	(*Zjeżdzam na osią pionową Z na pozycję chwytania i załączam ssawki*)		
	E_CapPreScrewer.ePicking:
		//Podjedź robotem w górę	
		mcCartesianZMoveAbsolute.Execute			:= TRUE;		
		mcCartesianZMoveAbsolute.Position			:= stParameters.lrPickZPosition;
		mcCartesianZMoveAbsolute.Acceleration		:= stParameters.lrPickerAcceleration;
		mcCartesianZMoveAbsolute.Deceleration		:= stParameters.lrPickerAcceleration;
		mcCartesianZMoveAbsolute.Velocity			:= stParameters.lrPickerSpeed;
		//Czekam na wykonanie ruchu
		IF mcCartesianZMoveAbsolute.Done THEN
			//Reset komendy ruchu osi
			mcCartesianZMoveAbsolute.Execute		:= FALSE;
			
			//Zeruje rejestry oraz załączanie ssawek
			 FOR i:=1 TO 4 DO
				 bCapSucker[i]						:= stParameters.bPickerActiv[i]; 
				 aCapPresence[i] 					:= FALSE;
			 END_FOR
	
			//Następny krok
			eRunningState							:= E_CapPreScrewer.eVacumCheckPart1;
		END_IF
	
	(*Sprawdzam czy zassane i jazda w górę*)	
	E_CapPreScrewer.eVacumCheckPart1:
		
		tonVacuumWatchdog.IN						:= TRUE;
		
		IF tonSuckedOk[1].Q = stParameters.bPickerActiv[1] AND tonSuckedOk[2].Q = stParameters.bPickerActiv[2]
			AND tonSuckedOk[3].Q = stParameters.bPickerActiv[3] AND tonSuckedOk[4].Q = stParameters.bPickerActiv[4] THEN
			tonVacuumWatchdog.IN					:= FALSE;
		
				FOR i:=1 TO 4 DO
					IF stParameters.bPickerActiv[i] AND stParameters.bStrawCatcherON AND NOT stMoverStatus.stSlotStatus[i].bTubePresent THEN
						bReject								:= TRUE;
						bTubeReject							:= TRUE;
						lrAxisZ_RejectOffset				:= 0.0;
					END_IF

					IF bMover1InPlacePos THEN
						diMover1VacuumRetry[i]		:= 0;
					ELSE
						diMover2VacuumRetry[i]		:= 0;
					END_IF	
				END_FOR 
				
			eRunningState 							:= E_CapPreScrewer.eVacumCheckPart2;
	
		ELSIF tonVacuumWatchdog.Q THEN
		
			FOR i:=1 TO 4 DO
				bCapSucker[i]							:= tonSuckedOk[i].Q;
				
				//robimy odrzut jeżeli zostanie wykryto brak słomki
				IF stParameters.bPickerActiv[i] AND stParameters.bStrawCatcherON AND NOT stMoverStatus.stSlotStatus[i].bTubePresent THEN
					bReject								:= TRUE;
					bTubeReject							:= TRUE;
					lrAxisZ_RejectOffset				:= 0.0;
				END_IF
				
						//Detekcja niepobranej nasadki --> odrzut aktywowany opcjonalnie z receptury
					IF stParameters.bPickerActiv[i] AND NOT tonSuckedOk[i].Q AND NOT stParameters.bVacuumDeactivate THEN
						bReject							:= SEL(stParameters.bRejectON, bReject, TRUE);
						lrAxisZ_RejectOffset			:= SEL(stParameters.bRejectON, lrAxisZ_RejectOffset, 13.0);	//offset dodatkowego zjazdu kartezjanem 
						
						IF bMover1InPlacePos THEN
							diMover1VacuumRetry[i]		:= diMover1VacuumRetry[i] + 1;
						ELSE	
							diMover2VacuumRetry[i]		:= diMover2VacuumRetry[i] + 1;
						END_IF
					ELSIF tonSuckedOk[i].Q OR stParameters.bVacuumDeactivate THEN
						IF 	bMover1InPlacePos THEN
							diMover1VacuumRetry[i]		:= 0;
						ELSE
							diMover2VacuumRetry[i]		:= 0;
						END_IF	
					END_IF	
	    	
			END_FOR
				tonVacuumWatchdog.IN					:= FALSE;
				eRunningState 							:= E_CapPreScrewer.eVacumCheckPart2;
	
		END_IF
		
		
	E_CapPreScrewer.eVacumCheckPart2:	
			
		//Jezeli nie jest przyssana zadna nasadka to pdjezdzamy na poz. ready oraz wystawiamy flage bMissingCaps
		IF bReject THEN
			Reject();
				IF bRejectDone THEN				
					eRunningState						:= E_CapPreScrewer.eReady;	
				END_IF		
		ELSIF NOT tonSuckedOk[1].Q AND NOT tonSuckedOk[2].Q AND NOT tonSuckedOk[3].Q AND NOT tonSuckedOk[4].Q THEN
			bCapSucker[1]							:= FALSE;
			bCapSucker[2]							:= False;
			bCapSucker[3]							:= False;
		    bCapSucker[4]							:= False;	
			mcCartesianZMoveAbsolute.Execute		:= TRUE;		
			mcCartesianZMoveAbsolute.Position		:= stParameters.lrTopZPosition;
			mcCartesianZMoveAbsolute.Acceleration	:= stParameters.lrPickerAcceleration;
			mcCartesianZMoveAbsolute.Deceleration	:= stParameters.lrPickerAcceleration;
			mcCartesianZMoveAbsolute.Velocity		:= stParameters.lrPickerSpeed;
			
			IF mcCartesianZMoveAbsolute.Done THEN
				bMissingCaps						:= TRUE;
				bCycleDone;
				mcCartesianZMoveAbsolute.Execute	:= FALSE;
				eRunningState						:= E_CapPreScrewer.eReady;	
			END_IF
			
		ELSE
			mcCartesianZMoveAbsolute.Execute		:= NOT stParameters.bVacuumDeactivate;		
			mcCartesianZMoveAbsolute.Position		:= stParameters.lrTopZPosition;
			mcCartesianZMoveAbsolute.Acceleration	:= SEL(GVL_Recipe.iCapSorterProductType = 0 ,stParameters.lrPickerAcceleration , 150.0);//stParameters.lrPickerAcceleration;
//			mcCartesianZMoveAbsolute.Acceleration	:= stParameters.lrPickerAcceleration;
			mcCartesianZMoveAbsolute.Deceleration	:= stParameters.lrPickerAcceleration;
			mcCartesianZMoveAbsolute.Velocity		:= stParameters.lrPickerSpeed;
			tonCapCatcher.IN						:= FALSE;
			
			IF mcCartesianZMoveAbsolute.Busy OR stParameters.bVacuumDeactivate THEN
				mcCartesianZMoveAbsolute.Execute		:= FALSE;
				eRunningState 							:= E_CapPreScrewer.eTransferingVertical; 
			END_IF
			
        
		END_IF		
			
			//przepisuje do rejestrów nakretki które kartezjan pobrał
			aCapPresence[1] := bCapSucker[1];
			aCapPresence[2] := bCapSucker[2];
			aCapPresence[3] := bCapSucker[3];
			aCapPresence[4] := bCapSucker[4];						

		
		
	(*Jazda w górę, zamknięcie łapek i załączenie jazdy w bok*)	
	E_CapPreScrewer.eTransferingVertical:
		
		IF NOT bCapSucker[1] OR NOT bCapSucker[2] OR NOT bCapSucker[3] OR NOT bCapSucker[4] THEN
            bCapBlow1						:= NOT bCapSucker[1];
            bCapBlow2						:= NOT bCapSucker[2];
            bCapBlow3						:= NOT bCapSucker[3];
            bCapBlow4						:= NOT bCapSucker[4];						
			bCapsBlowON						:= TRUE;
		END_IF
		
		//Kleją się kulki 
		IF NOT stParameters.bVacuumDeactivate THEN					
			IF CartesianZAxisRef.NcToPlc.ActPos > stParameters.lrPickZPosition + 10.0 THEN
				mcCartesianZMoveAbsolute2.Execute		:= NOT stParameters.bVacuumDeactivate;		
				mcCartesianZMoveAbsolute2.Position		:= stParameters.lrTopZPosition;
				mcCartesianZMoveAbsolute2.Acceleration	:= stParameters.lrPickerAcceleration;
				mcCartesianZMoveAbsolute2.Deceleration	:= stParameters.lrPickerAcceleration;
				mcCartesianZMoveAbsolute2.Velocity		:= stParameters.lrPickerSpeed;
			END_IF
		END_IF


		IF CartesianZAxisRef.NcToPlc.ActPos > stParameters.lrCapCatcherZPosition OR (CartesianZAxisRef.NcToPlc.ActPos > stParameters.lrTopZPosition - stParameters.lrBendingDistance) THEN
			bCapCatcher1							:= TRUE;
			bCapCatcher2							:= true;
			bCapCatcher3							:= true;
			bCapCatcher4							:= true;
			tonCapCatcher.IN						:= stParameters.bVacuumDeactivate;
		END_IF	
		
		mcCartesianZMoveAbsolute.Execute		:= tonCapCatcher.Q;	
		
		//Dodać sprawdzenie czy gotowy chwytak słomek !!!!!
		//Sprawdzenie pozycji osi pionowej Z i czy wysunięty siłownik chwytaka słomek
		IF ((CartesianZAxisRef.NcToPlc.ActPos > stParameters.lrTopZPosition - stParameters.lrBendingDistance) OR
			mcCartesianZMoveAbsolute.Done) AND (tonStrawCatcherOut.Q OR NOT stParameters.bStrawCatcherON) THEN
			//Jedź osią poziomą X na pozycję pick
				mcCartesianZMoveAbsolute2.Execute		:= FALSE;
				bCapsBlowON								:= FALSE;
				eRunningState 							:= E_CapPreScrewer.eTransferingHorizontal;
				tonCapCatcher.IN						:= FALSE;
		END_IF
	
	(*Przejazd w poziomie*)	
	E_CapPreScrewer.eTransferingHorizontal:	
	
			bCapCatcher1							:= TRUE;//bCapSucker1;
			bCapCatcher2							:= TRUE;//bCapSucker2;
			bCapCatcher3							:= TRUE;//bCapSucker3;
			bCapCatcher4							:= TRUE;//bCapSucker4;
	
		mcCartesianYMoveAbsolute.Position			:= stParameters.lrPlaceYPosition;
		mcCartesianYMoveAbsolute.Acceleration		:= stParameters.lrPickerAcceleration;
		mcCartesianYMoveAbsolute.Deceleration		:= stParameters.lrPickerAcceleration;
		mcCartesianYMoveAbsolute.Velocity			:= stParameters.lrPickerSpeed;
		mcCartesianYMoveAbsolute.Execute			:= TRUE;
		
		IF (CartesianYAxisRef.NcToPlc.ActPos > 200.0 (*stParameters.lrPlaceYPosition - stParameters.lrBendingDistance*)) OR
			mcCartesianYMoveAbsolute.Done AND NOT mcCartesianZMoveAbsolute.Execute THEN			

			//Podjedź robotem w dól	
			mcCartesianZMoveAbsolute.Execute			:= TRUE;		
			mcCartesianZMoveAbsolute.Position			:= stParameters.lrCartesianCatchZPosition;
			mcCartesianZMoveAbsolute.Acceleration		:= stParameters.lrPickerAcceleration;
			mcCartesianZMoveAbsolute.Deceleration		:= stParameters.lrPickerAcceleration;
			mcCartesianZMoveAbsolute.Velocity			:= stParameters.lrPickerSpeed;
		END_IF
		
		//Jak obie pozycje osiągnięte 
		IF mcCartesianZMoveAbsolute.Done THEN
			mcCartesianZMoveAbsolute.Execute		:= FALSE;
		END_IF
			
		//Jak ak obie pozycje osiągnięte to zamykamy chwytaki i następny krok
		IF stParameters.bStrawCatcherON AND CartesianYAxisRef.NcToPlc.ActPos >= stParameters.lrPlaceYPosition THEN
			//Zamknij chwytaki słomek
			bStrawCatchersOpen						:= FALSE;
			bStrawCatchersClose						:= TRUE;	
		END_IF
		
			
		IF  mcCartesianYMoveAbsolute.Done AND mcCartesianZMoveAbsolute.Done THEN
			//Reset komendy ruchu osi
			mcCartesianYMoveAbsolute.Execute		:= FALSE;
			mcCartesianZMoveAbsolute.Execute		:= FALSE;
			
				//Ustaw pozycję wirtualnej osi tak samo jak na osi Z
			fbVirtualAxis.fPosition						:=  CartesianZAxisRef.NcToPlc.ActPos;//CartesianZAxisRef.NcToPlc.ActPos - GVL_Recipe.lrCapSorterCapNeckHightShow - GVL_Recipe.lrCapSorterPreScrewerCheckValveShow;
			fbVirtualAxis.SetPosAbsClearLag(bExecute	:= TRUE);
				
				IF fbVirtualAxis.pSetPos.Busy THEN
					//Następny krok
					eRunningState						:= E_CapPreScrewer.eVerticalDownToCatchPos;	
				END_IF
		END_IF		
		
	(*Przejazd w dól do pozycji chwytanija rurki*)		
	E_CapPreScrewer.eVerticalDownToCatchPos:
		fbVirtualAxis.SetPosAbsClearLag(bExecute				:= FALSE);
		
		//Jak ak obie pozycje osiągnięte to zamykamy chwytaki i następny krok
		IF stParameters.bStrawCatcherON THEN
			//Zamknij chwytaki słomek
			bStrawCatchersOpen						:= FALSE;
			bStrawCatchersClose						:= TRUE;	
		END_IF
				
		IF tonPlacePermission.Q AND ((bCapCatcher1 OR NOT bCapCatcher1) AND (bCapCatcher2  OR NOT bCapCatcher2) AND
									(bCapCatcher3  OR NOT bCapCatcher3) AND(bCapCatcher4  OR NOT bCapCatcher4)) AND (tonStrawCatcher1Close.Q OR NOT stParameters.bStrawCatcherON) THEN				
				bCapCatcher1						:= TRUE;
				bCapCatcher2						:= TRUE;
				bCapCatcher3						:= TRUE;
				bCapCatcher4						:= TRUE;						
				eRunningState						:= E_CapPreScrewer.eAxisGearIn;
		END_IF
		
	
	E_CapPreScrewer.eAxisGearIn:
		fbGearInCatcherAxis.Enable						:= stParameters.bStrawCatcherON;
		fbGearInCatcherAxis.GearRatio					:= 1;
		
		fbGearInPos.Execute								:= NOT fbGearInPos.Active;
		fbGearInPos.MasterSyncPosition					:= stParameters.lrCartesianCatchZPosition - (stParameters.lrCapHight - GVL_Recipe.lrCapSorterCapNeckHightShow - GVL_Recipe.lrCapSorterPreScrewerCheckValveShow);//10
		fbGearInPos.SlaveSyncPosition					:= stParameters.lrCartesianCatchZPosition - 15;//15
		
		
		
			IF (fbGearInCatcherAxis.InGear OR NOT stParameters.bStrawCatcherON) AND fbGearInPos.Active AND (tonStrawCatcher1Close.Q (*AND tonStrawCatcher2Close.Q*)
				OR (bStrawCatcherOpen1 AND bStrawCatcherOpen2 AND bStrawCatcherOpen3 AND bStrawCatcherOpen4))  THEN
					fbGearInCatcherAxis.Enable			:= FALSE;
					fbGearInPos.Execute					:= FALSE;
						IF stParameters.bStrawCatcherON THEN
							eRunningState				:= E_CapPreScrewer.ePositionOverBottle;	
							//fbVirtualAxis.fPosition		:= stParameters.lrCartesianCatchZPosition -(CatcherAxisRef.NcToPlc.ActPos - (stParameters.lrBottleHight - stParameters.lrCatcherHightSV - 35));//40mm- offset między łapkami słomek a chwytakami butelek
							lrPreScrewerAxisSavedPosition	:= stParameters.lrCartesianCatchZPosition -(CatcherAxisRef.NcToPlc.ActPos - (stParameters.lrBottleHight - stParameters.lrCatcherHightSV - 35));
							fbVirtualAxis.fPosition		:= (stParameters.LrCheckStrawCatcherActuatorZPosition - (fbGearInPos.SlaveSyncPosition - fbGearInPos.MasterSyncPosition));
						ELSE                            
							eRunningState				:= E_CapPreScrewer.ePlacing;	
						END_IF					
			END_IF		
	
	E_CapPreScrewer.ePositionOverBottle:
		fbVirtualAxis.fVelocity							:= SEL(stParameters.lrCatcherSpeed > 1094.0, stParameters.lrCatcherSpeed, 1094.0 );       						
			
		
		//IF fbVirtualAxis.Axis.NcToPlc.ActPos <= fbVirtualAxis.fPosition	+ 10.0 OR (CatcherAxisRef.NcToPlc.ActPos <= 5.0) THEN
		IF fbVirtualAxis.Axis.NcToPlc.ActPos <= lrPreScrewerAxisSavedPosition	+ 10.0 OR (CatcherAxisRef.NcToPlc.ActPos <= 5.0) THEN
			fbGearInCatcherAxis.GearRatio				:= 0.0000000000000000000000000000000000000000000000000000000000001;		
			fbGearOutCatcherAxis.Execute				:= CatcherAxisRef.Status.Coupled;
			mcCatcherStop.Execute						:= 	NOT CatcherAxisRef.Status.Coupled ;
			bVirtualMove								:= FALSE;
		ELSE
			bVirtualMove								:= TRUE;	
		END_IF 
		
		IF NOT CatcherAxisRef.Status.Coupled AND (NOT CatcherAxisRef.Status.Moving OR mcCatcherStop.Busy) THEN
			eRunningState							:= E_CapPreScrewer.eCatching;	
		END_IF
	
	
	//Sprawdzanie czy chwytaki zamknięte i opuszczenie chwytaków do dolnej pozycji
	E_CapPreScrewer.eCatching:
		fbVirtualAxis.fPosition							:= (stParameters.LrCheckStrawCatcherActuatorZPosition - (fbGearInPos.SlaveSyncPosition - fbGearInPos.MasterSyncPosition));// - stParameters.lrStrawInsertDistance);	//Pozycja sprawdzania cofnięcia krabów
		fbVirtualAxis.fVelocity							:= SEL(stParameters.lrCatcherSpeed > 1094.0, stParameters.lrCatcherSpeed, 1094.0 );       						
		bVirtualMove									:= TRUE;					
	
			//Otwórz chwytaki słomek
		IF CartesianZAxisRef.NcToPlc.ActPos <= stParameters.lrStrawCatcherZPosition THEN		
			bStrawCatchersOpen							:= TRUE;
			bStrawCatchersClose							:= FALSE;
			
				IF tonStrawCatcher1Open.Q AND tonStrawCatcher2Open.Q AND tonStrawCatcher3Open.Q AND tonStrawCatcher4Open.Q THEN																				
					//Cofnij chwytaki słomek
					bStrawCatcherActuatorIn				:= TRUE;
					bStrawCatcherActuatorOut			:= FALSE;				
				END_IF	
		ELSE
			fbGearInCatcherAxis.GearRatio				:= F_Scaling((CatcherAxisRef.NcToPlc.ActPos*10), 0.0, 10.0, 0.0, 1.0);
			fbGearInCatcherAxis.GearRatio				:= SEL(fbGearInCatcherAxis.GearRatio>1.0, fbGearInCatcherAxis.GearRatio, 1.0);	
		END_IF		
						
				IF bStrawCatcherIn THEN
					fbGearOutCatcherAxis.Execute		:= FALSE;
					mcCatcherStop.Execute				:= FALSE;
					bVirtualMove						:= FALSE;	
					eRunningState						:= E_CapPreScrewer.ePlacing;
				END_IF		
			
		//END_IF
	


	
	//Czekaj aż chwytak słomek dojedzie do dołu i zacznij ruch osi pionowej Z
	E_CapPreScrewer.ePlacing:		
		IF stParameters.lrScrewFinding > 0 THEN
			eRunningState								:= E_CapPreScrewer.eFinding;
		ELSE
			lrPreScrewerAxisSavedPosition				:= PreScrewerAxisRef.NcToPlc.ActPos;	//zapisywanie pozycji przed zakrecaniem		
			fbVirtualAxis.fPosition						:= SEL(stParameters.bStrawCatcherON, stParameters.lrScrewerStartZPosition, stParameters.lrScrewerStartZPosition - (fbGearInPos.SlaveSyncPosition - fbGearInPos.MasterSyncPosition));//stParameters.lrPlaceZPosition, stParameters.lrPlaceZPosition - (fbGearInPos.SlaveSyncPosition - fbGearInPos.MasterSyncPosition));//stParameters.lrStrawInsertDistance);
			fbVirtualAxis.fVelocity						:= SEL(stParameters.lrCatcherSpeed > 1094.0, stParameters.lrCatcherSpeed, 1094.0 );    
			bVirtualMove								:= TRUE;
			
			eRunningState								:= E_CapPreScrewer.ePreScrewing;
		END_IF
	
	E_CapPreScrewer.eFinding:
		fbVirtualAxis.fPosition							:= SEL(stParameters.bStrawCatcherON, stParameters.lrScrewerStartZPosition, stParameters.lrScrewerStartZPosition - (fbGearInPos.SlaveSyncPosition - fbGearInPos.MasterSyncPosition));// stParameters.lrScrewerStartZPosition-stParameters.lrStrawInsertDistance);
		fbVirtualAxis.fVelocity							:= SEL(stParameters.lrCatcherSpeed > 1094.0, stParameters.lrCatcherSpeed, 1094.0 );
		fbVirtualAxis.fAcceleration						:= stParameters.lrCatcherAcceleration; 
		fbVirtualAxis.fDeceleration						:= stParameters.lrCatcherAcceleration; 
		fbVirtualAxis.fJerk								:= stParameters.lrCatcherJerk;        		
			                                            
		bVirtualMove									:= TRUE;
		                                                
			IF ABS(fbVirtualAxis.Axis.NcToPlc.ActPos - fbVirtualAxis.fPosition) <= 0.5 THEN              
				bCapSucker[1]								:= FALSE;
				bCapSucker[2]								:= FALSE;
				bCapSucker[3]								:= FALSE;
				bCapSucker[4]								:= FALSE;
    	                                                
				mcPreScrewerMoveRelative.Distance		:= stParameters.lrScrewFinding * -1.0;
				mcPreScrewerMoveRelative.Acceleration	:= stParameters.lrScrewAcceleration;
				mcPreScrewerMoveRelative.Deceleration	:= stParameters.lrScrewAcceleration;
				mcPreScrewerMoveRelative.Velocity		:= stParameters.lrScrewSpeed;
				mcPreScrewerMoveRelative.Execute		:= TRUE;
			END_IF
			
					IF mcPreScrewerMoveRelative.Done OR ABS(PreScrewerAxisRef.NcToPlc.PosDiff) > 60.0 OR mcPreScrewerMoveRelative.Error THEN
						bVirtualMove							:= FALSE;
						mcPreScrewerMoveRelative.Execute		:= FALSE;
						eRunningState							:= E_CapPreScrewer.ePreScrewing;
					END_IF	
	
	E_CapPreScrewer.ePreScrewing:

	IF ABS(fbVirtualAxis.Axis.NcToPlc.ActPos - fbVirtualAxis.fPosition)<=0.1 THEN
		bVirtualMove											:= FALSE;
		
		IF NOT	CartesianZAxisRef.Status.Coupled THEN
			eRunningState				:= E_CapPreScrewer.eScrewing;
			mcCartesianZStop.Execute	:= FALSE;
			fbGearOutAxisZ.Execute		:= FALSE;
		ELSE
			fbGearOutAxisZ.Execute		:= TRUE;
			mcCartesianZStop.Execute	:= CartesianZAxisRef.Status.Moving;
		END_IF	
	END_IF
		
	
	
	E_CapPreScrewer.eScrewing:
	
			fbGearInAxisZ_Screwer.Execute			:= NOT CartesianZAxisRef.Status.Coupled AND NOT mcCartesianZStop.Busy;
			fbGearInAxisZ_Screwer.RatioNumerator 	:= (GVL_Recipe.lrCapSorterPreScrewerThreadPitchShow	* GVL_Recipe.lrCapSorterPreScrewerMultipleStartThreadShow * (-1));
			fbGearInAxisZ_Screwer.RatioDenominator	:= 360;
		
			IF CartesianZAxisRef.Status.Coupled THEN	//+8
						mcPreScrewerMoveRelative.Execute		:= TRUE;
						mcPreScrewerMoveRelative.Distance		:= stParameters.lrScrewDistance;
						mcPreScrewerMoveRelative.Acceleration	:= stParameters.lrScrewAcceleration;
						mcPreScrewerMoveRelative.Deceleration	:= stParameters.lrScrewAcceleration;
						mcPreScrewerMoveRelative.Velocity		:= stParameters.lrScrewSpeed;	
						eRunningState							:= E_CapPreScrewer.eFinished;	
			END_IF
	
	//Kończenie cyklu zakręcania - otwarcie chwytaka
	E_CapPreScrewer.eFinished:		
	
		IF PreScrewerAxisRef.NcToPlc.PosDiff > 100.0 OR mcPreScrewerMoveRelative.Done THEN
//			bBottleCatcherCatchTemp							:= FALSE;	
			bCapCatcher1									:= FALSE;
		 	bCapCatcher2									:= FALSE;
		 	bCapCatcher3									:= FALSE;
		 	bCapCatcher4									:= FALSE;
			mcPreScrewerMoveRelative.Execute				:= FALSE;
			bVirtualMove									:= FALSE;
			bCapBlow1										:= bCapSucker[1];
            bCapBlow2										:= bCapSucker[2];
            bCapBlow3										:= bCapSucker[3];
            bCapBlow4										:= bCapSucker[4];
			bCapSucker[1]									:= FALSE;
			bCapSucker[2]									:= FALSE;
			bCapSucker[3]									:= FALSE;
			bCapSucker[4]									:= FALSE;								
			
				IF PreScrewerAxisRef.Status.Moving THEN
					mcPreScrewerStop.Execute				:=	 TRUE;					
				ELSE
					lrAxisZSavedPosition					:= CartesianZAxisRef.NcToPlc.ActPos;
					mcPreScrewerStop.Execute				:= FALSE;
					fbGearInCatcherAxis.Enable				:= FALSE;
					eRunningState							:= E_CapPreScrewer.eGearOut;
				END_IF	
		END_IF
		
	E_CapPreScrewer.eGearOut:
		fbGearOutAxisZ.Execute								:= TRUE;
		fbGearOutCatcherAxis.Execute						:= TRUE;
	
			IF NOT CartesianZAxisRef.Status.Coupled AND NOT CatcherAxisRef.Status.Coupled THEN
				fbGearOutAxisZ.Execute						:= FALSE;
				fbGearOutCatcherAxis.Execute				:= FALSE;
				eRunningState								:= E_CapPreScrewer.eReturning1;
			END_IF
	
	//Powrót na górną pozycję
	E_CapPreScrewer.eReturning1:
	
		tonWaitInPlacePos.IN						:= TRUE;
		mcPreScrewerStop.Execute					:= TRUE;		

		IF tonWaitInPlacePos.Q THEN
			

		
			tonWaitInPlacePos.IN					:= FALSE;
//			bBottleCatcherCatchTemp					:= FALSE;		
			mcPreScrewerStop.Execute				:= FALSE;
			mcCartesianZMoveAbsolute.Execute		:= TRUE;
			mcCartesianZMoveAbsolute.Position		:= stParameters.lrTopZPosition;
			mcCartesianZMoveAbsolute.Acceleration	:= SEL(GVL_Recipe.iCapSorterProductType = 0 ,stParameters.lrPickerAcceleration , 150.0);
//			mcCartesianZMoveAbsolute.Acceleration	:= stParameters.lrPickerAcceleration;
			mcCartesianZMoveAbsolute.Deceleration	:= stParameters.lrPickerAcceleration;
			mcCartesianZMoveAbsolute.Velocity		:= stParameters.lrPickerSpeed;
			
			IF mcCartesianZMoveAbsolute.Busy THEN
				mcCartesianZMoveAbsolute.Execute		:= FALSE;
				eRunningState							:= E_CapPreScrewer.eReturning2;
			END_IF
			
		END_IF
		

		
	//Powrót po osi X	
	E_CapPreScrewer.eReturning2:
		bBottleCatcherCatchTemp					:= FALSE;
		bCapsBlowON								:= CartesianZAxisRef.NcToPlc.ActPos > lrAxisZSavedPosition + 10.0;
		
		IF CartesianZAxisRef.NcToPlc.ActPos > stParameters.lrScrewerStartZPosition + 15.0 THEN
			mcCartesianZMoveAbsolute2.Execute		:= TRUE;
			mcCartesianZMoveAbsolute2.Position		:= stParameters.lrTopZPosition;
			mcCartesianZMoveAbsolute2.Acceleration	:= stParameters.lrPickerAcceleration;
			mcCartesianZMoveAbsolute2.Deceleration	:= stParameters.lrPickerAcceleration;
			mcCartesianZMoveAbsolute2.Velocity		:= stParameters.lrPickerSpeed;			
		END_IF
	
		IF (CartesianZAxisRef.NcToPlc.ActPos > stParameters.lrTopZPosition - stParameters.lrBendingDistance) OR
			mcCartesianZMoveAbsolute.Done THEN
			mcCatcherMoveAbsolute.Execute			:= TRUE;		
			mcCatcherMoveAbsolute.Position			:= stParameters.lrCatcherCatchingPosition;
			mcCatcherMoveAbsolute.Acceleration		:= stParameters.lrCatcherAcceleration;
			mcCatcherMoveAbsolute.Deceleration		:= stParameters.lrCatcherAcceleration;
			mcCatcherMoveAbsolute.Velocity			:= stParameters.lrCatcherSpeed;

//SEL(P190_CapFeeder.stMover2Status.bInPlacePosition, GVL_Recipe.lrCapSorterPreScrewerPickXMover1PositionShow, GVL_Recipe.lrCapSorterPreScrewerPickXMover2PositionShow

			
			//Jedź osią poziomą X na pozycję pick
			mcCartesianYMoveAbsolute.Execute		:= TRUE;
			{warning 'Przerobić, dodać parametry obu pozycji wózków do struktury parametrów, FB_CapPreScrewer.Running --> 624'}
			mcCartesianYMoveAbsolute.Position		:= SEL(bMover1InPickPos, GVL_Recipe.lrCapSorterPreScrewerPickXMover1PositionShow, GVL_Recipe.lrCapSorterPreScrewerPickXMover2PositionShow);
			mcCartesianYMoveAbsolute.Acceleration	:= stParameters.lrPickerAcceleration;
			mcCartesianYMoveAbsolute.Deceleration	:= stParameters.lrPickerAcceleration;
			mcCartesianYMoveAbsolute.Velocity		:= stParameters.lrPickerSpeed;
			//Ustaw obracarkę do pozycji początkowej
			
			mcPreScrewerMoveRelative.Distance		:= -1 * DINT_TO_LREAL(LREAL_TO_DINT(PreScrewerAxisRef.NcToPlc.SetPos) MOD 360); 
			mcPreScrewerMoveRelative.Execute		:= mcPreScrewerMoveRelative.Distance<>0 AND NOT mcPreScrewerMoveRelative.Error;
			mcPreScrewerMoveRelative.Acceleration	:= stParameters.lrScrewAcceleration;
			mcPreScrewerMoveRelative.Deceleration	:= stParameters.lrScrewAcceleration;
			mcPreScrewerMoveRelative.Velocity		:= stParameters.lrScrewSpeed;
			
		END_IF
		IF CartesianZAxisRef.NcToPlc.ActPos > stParameters.lrPlaceZPosition + 20 THEN
			bPlaceDone								:= TRUE;
		END_IF
		IF (*bPlaceDone AND*) mcCartesianYMoveAbsolute.Done AND mcCartesianZMoveAbsolute2.Done AND
			 mcCatcherMoveAbsolute.Done THEN
			 IF mcPreScrewerMoveRelative.Distance=0 OR mcPreScrewerMoveRelative.Done THEN
				mcCartesianYMoveAbsolute.Execute		:= FALSE;
 				mcCartesianZMoveAbsolute.Execute		:= FALSE;
				mcCartesianZMoveAbsolute2.Execute		:= FALSE;
				mcCatcherMoveAbsolute.Execute			:= FALSE;
				mcPreScrewerMoveRelative.Execute		:= FALSE;
				eRunningState				:= E_CapPreScrewer.eDone;
			END_IF
		END_IF
		
		//Dodatkowy przedmuch ssawek
		(*IF (CartesianZAxisRef.NcToPlc.ActPos > (stParameters.lrPlaceZPosition + stParameters.lrHeightAdditionalBlow)) THEN
			bAdditionalBlow							S= NOT tonBlowOFF.IN;	
		
			IF NOT bAdditionalBlow THEN
				bCapsBlowON							R= tonBlowOFF.Q;
			END_IF

			bCapsBlowON								S= bAdditionalBlow;
			bCapBlow1 := bCapBlow2 := bCapBlow3 := bCapBlow4 := bAdditionalBlow;
		END_IF*)
			
	E_CapPreScrewer.eDone:
		mcPreScrewerStop.Execute			:= TRUE;
	
		IF mcPreScrewerStop.Done THEN
			mcPreScrewerStop.Execute			:= FALSE;
			bAdditionalBlow						:= FALSE;
			bCycleNotDone						:= FALSE;
			bCapsBlowON							:= FALSE;
			bPlaceDone							:= TRUE;
			bCycleDone							:= TRUE;
			eState								:= E_Station.eDone;
			eRunningState						:= E_CapPreScrewer.eReady;	
		END_IF	

	(*Cykl nie zakończony - przerwany - chyba nie potrzebny*)
	E_CapPreScrewer.eNotDone:
		bCapsBlowON							:= FALSE;
		eState								:= E_Station.eDone;
		eRunningState						:= E_CapPreScrewer.eReady;




END_CASE

tonCapCatcher(PT := T#60MS);
END_ACTION

ACTION Signals:
rtChoseRecipe(CLK := stCommandsIn.bChoseRecipe);
rtAxisZMoving(CLK := CartesianZAxisRef.Status.Moving);
bHomingWithoutJiesang	R= rtChoseRecipe.Q;

//Filtry sygnałów z czujników 
tonSuckedOk[1](IN:=bCapSucker[1] AND (stParameters.bVacuumDeactivate OR bCapSuckerVacumOk1), PT:=T#4MS);
tonSuckedOk[2](IN:=bCapSucker[2] AND (stparameters.bvacuumDeactivate OR bCapSuckerVacumOk2), PT:=T#4MS);
tonSuckedOk[3](IN:=bCapSucker[3] AND (stparameters.bvacuumDeactivate OR bCapSuckerVacumOk3), PT:=T#4MS);
tonSuckedOk[4](IN:=bCapSucker[4] AND (stparameters.bvacuumDeactivate OR bCapSuckerVacumOk4), PT:=T#4MS);

tonStrawCatcherIn(In:=bStrawCatcherIn, PT:=T#4MS); 
tonStrawCatcherOut(In:=bStrawCatcherOut, PT:=T#4MS);

tonStrawCatcher1Open(In:=  bStrawCatcherOpen1, PT:=T#0MS); 
tonStrawCatcher2Open(In:=  bStrawCatcherOpen2, PT:=T#0MS); 
tonStrawCatcher3Open(In:=  bStrawCatcherOpen3, PT:=T#0MS); 
tonStrawCatcher4Open(In:=  bStrawCatcherOpen4, PT:=T#0MS); 

tonStrawCatcher1Close(In:=NOT bStrawCatcherOpen1 OR bStrawCatchersClose, PT:=T#120MS); 
tonStrawCatcher2Close(In:=NOT bStrawCatcherOpen2, PT:=T#0MS); 
tonStrawCatcher3Close(In:=NOT bStrawCatcherOpen3, PT:=T#0MS); 
tonStrawCatcher4Close(In:=NOT bStrawCatcherOpen4, PT:=T#0MS); 	

tonCapCatcher1Open(IN:= NOT bCapCatcher1, PT := T#50MS);

tonBlowOFF.PT := SEL(eRunningState = E_CapPreScrewer.eTransferingVertical, T#250MS, T#2S);
tonBlowOFF(In:=bCapsBlowON); 	//250ms //dp bylo 50
tonBlowerON[1](In:=bCapsBlowON, PT:=T#0MS); //timery na załączanie kolejnych cewek
tonBlowerON[2](In:=bCapsBlowON, PT:=T#4MS); (*T#15MS*)
tonBlowerON[3](In:=bCapsBlowON, PT:=T#8MS); 
tonBlowerON[4](In:=bCapsBlowON, PT:=T#12MS);

bCapBlower1 			:= (*tonBlowerON[1].Q AND*) bCapsBlowON AND NOT tonBlowOFF.Q AND (bCapBlow1 (*OR aCapPresence[1]*));
bCapBlower2 			:= (*tonBlowerON[2].Q AND*) bCapsBlowON AND NOT tonBlowOFF.Q AND (bCapBlow2 (*OR aCapPresence[2]*));
bCapBlower3 			:= (*tonBlowerON[3].Q AND*) bCapsBlowON AND NOT tonBlowOFF.Q AND (bCapBlow3 (*OR aCapPresence[3]*));
bCapBlower4 			:= (*tonBlowerON[4].Q AND*) bCapsBlowON AND NOT tonBlowOFF.Q AND (bCapBlow4 (*OR aCapPresence[4]*));
	
tonPlacePermission(IN 	:= bPlacePermission, PT:=T#30MS); 
rtPlacePermission(CLk 	:= tonPlacePermission.Q);
rtRun(CLK	:= bRun);
//Żądanie zamknięcia chwytaków
IF rtPlacePermission.Q THEN
	bBottleCatcherCatchTemp			:= TRUE;
END_IF

//Przewidywane zatrzymanie, wymuś bazowanie jezeli kartezjan nie bedzie na tych pozycjach!!!!!
bCartesianInReadyPos	:= (eRunningState = E_CapPreScrewer.eReady) OR
							(eRunningState = E_CapPreScrewer.eVerticalDownToCatchPos);
	
//Flagi pomocnicze dla bazowania- AxisY jest na pozycji
bAxisYInPosition	:= ABS(mcCartesianYMoveAbsolute.Position - CartesianYAxisRef.NcToPlc.ActPos) < 10.0;

//Flagi pomocnicze dla bazowania- AxisZ jest na pozycji 1
bAxisZInPosition1 := NOT CartesianZAxisRef.Status.Moving AND ABS(mcCartesianZMoveAbsolute.Position - CartesianZAxisRef.NcToPlc.ActPos) < 10.0;

//Flagi pomocnicze dla bazowania- AxisZ jest na pozycji 2
bAxisZInPosition2	:= NOT CartesianZAxisRef.Status.Moving AND ABS(mcCartesianZMoveAbsolute2.Position - CartesianZAxisRef.NcToPlc.ActPos) < 10.0;

//Oś Z jest na pozycji
bAxisZInPosition := bAxisZInPosition1 OR bAxisZInPosition2;
															
IF tonBlowOFF.Q THEN
	bCapsBlowON 							:= FALSE;
	bCapBlow1								:= FALSE;
	bCapBlow2								:= FALSE;
	bCapBlow3								:= FALSE;
	bCapBlow4								:= FALSE;
END_IF

bAxisYSafePos			:= CartesianYAxisRef.NcToPlc.ActPos > 250.0;
bCartesianSafePos			:= (CartesianZAxisRef.NcToPlc.ActPos >= 310.0) OR bAxisYSafePos;

//Monitoring utraconych nasadek, sprawdzamy tylko gdy odjeżdżamy do poz. place oraz mamy zamknąć wings'y
IF eRunningState > 5 AND eRunningState < 30 THEN
	bCapLost[1]								:= NOT bCapCatcher1  AND stParameters.bPickerActiv[1]; 
	bCapLost[2]								:= NOT bCapCatcher2  AND stParameters.bPickerActiv[2]; 
	bCapLost[3]								:= NOT bCapCatcher3  AND stParameters.bPickerActiv[3]; 
	bCapLost[4]								:= NOT bCapCatcher4  AND stParameters.bPickerActiv[4]; 
	bAnyCapLost								:= bCapLost[1] OR bCapLost[2] OR bCapLost[3] OR bCapLost[4];
ELSE
	bCapLost[1]								:= FALSE;
    bCapLost[2]								:= False;
    bCapLost[3]								:= False;
    bCapLost[4]								:= False;
    bAnyCapLost								:= False;
END_IF

bAnyCapPresence		:= (bCapSuckerVacumOk1 OR bCapCatcher1 OR bCapSuckerVacumOk2 OR bCapCatcher2 OR 
						bCapSuckerVacumOk3 OR bCapCatcher3 OR bCapSuckerVacumOk4 OR bCapCatcher4);

bAxisZInHomePos 	:= ABS(CartesianZAxisRef.NcToPlc.ActPos - 420.0) <= 1.0;
bAxisZInTopPos		:= ABS(CartesianZAxisRef.NcToPlc.ActPos - stParameters.lrTopZPosition) <= 1.0;
bAxisYInHomePos		:= ABS(CartesianYAxisRef.NcToPlc.ActPos - stParameters.lrPickYPosition) <= 1.0;
bStrawCatcherLiftInHomePos := tonStrawCatcherLiftInHomePos.Q;
bCartesianInHomePos	:= bAxisZInHomePos AND bAxisYInHomePos;
bCartesianInTopPos  := bAxisZInTopPos AND bAxisYInHomePos;

//Kąt początkowy zakręcarki
diPreSCrewerHomePos	:= SEL(GVL_Recipe.bCapSorterPreScrewerPoundedInCap, 0, 90);

//Monitorowanie momentu na osiach
CartesianYAxisRef.NcToPlc.ActTorque;
CartesianZAxisRef.NcToPlc.ActTorque;
CatcherAxisRef.NcToPlc.ActTorque;


bCapScrewed		:= (eLastRunningState = E_CapPreScrewer.eFinding OR eLastRunningState = E_CapPreScrewer.eFindingStop
					OR eLastRunningState = E_CapPreScrewer.eScrewing OR eLastRunningState = E_CapPreScrewer.eFinished
					OR eLastRunningState = E_CapPreScrewer.eReturning1);


tonStrawCatcherLiftInHomePos(IN := ABS(GVL_VIS.lrCapSorterPreScrewerCatcherStationHeightCV-stParameters.lrCatcherHightSV) <= 1.0, PT := T#3S);

FOR i:=1 TO 4 DO
	arrVacuumStatus[i] := tonSuckedOk[i].Q OR (NOT bCapSucker[i] AND NOT stParameters.bPickerActiv[i]);
END_FOR


bAllSlotsVacuumStatus	:= arrVacuumStatus[1] AND arrVacuumStatus[2] AND arrVacuumStatus[3] AND arrVacuumStatus[4];
END_ACTION

ACTION Simulation:
tonVacuumWatchdog(PT	:= stParameters.tTimeVacuumWatchdog);
bStopAllowed	:= iSimulationCase = 0;

CASE iSimulationCase OF
	0:
			IF NOT bCycleDone AND NOT bCycleNotDone THEN  
				IF bRun THEN 
				iRejectCase					:= 0;
				bRejectDone					:= FALSE;
				bReject						:= FALSE;
				bTubeReject					:= FALSE;
				
				//Przygotuj do cyklu - otwórz chwytaki
				bCapCatcher1				:= FALSE;
				bCapCatcher2				:= FALSE;
				bCapCatcher3				:= FALSE;
				bCapCatcher4				:= FALSE;
	
				//Wyłącz ssawki
				bCapSucker[1]				:= FALSE;
				bCapSucker[2]				:= FALSE;
				bCapSucker[3]				:= FALSE;
				bCapSucker[4]				:= FALSE;
				//Wyłącz odmuchy
				bCapBlower1					:= FALSE;
				bCapBlower2					:= FALSE;
				bCapBlower3					:= FALSE;
				bCapBlower4					:= FALSE;
				bCapsBlowON					:= FALSE;
				//Otwórz chwytaki słomek
				bStrawCatchersOpen			:= TRUE;
				bStrawCatchersClose			:= FALSE;
				//Cofnij chwytaki słomek
				bStrawCatcherActuatorIn		:= TRUE;
				bStrawCatcherActuatorOut	:= FALSE;
				
					IF tonStrawCatcherIn.Q THEN	
											
						mcCartesianZMoveAbsolute.Execute		:= TRUE;		
						mcCartesianZMoveAbsolute.Position		:= stParameters.lrTopZPosition;
						mcCartesianZMoveAbsolute.Acceleration	:= stParameters.lrPickerAcceleration;
						mcCartesianZMoveAbsolute.Deceleration	:= stParameters.lrPickerAcceleration;
						mcCartesianZMoveAbsolute.Velocity		:= stParameters.lrPickerSpeed;
						
						mcCatcherMoveAbsolute.Execute			:= TRUE;		
						mcCatcherMoveAbsolute.Position			:= stParameters.lrCatcherCatchingPosition;
						mcCatcherMoveAbsolute.Acceleration		:= stParameters.lrCatcherAcceleration;
						mcCatcherMoveAbsolute.Deceleration		:= stParameters.lrCatcherAcceleration;
						mcCatcherMoveAbsolute.Velocity			:= stParameters.lrCatcherSpeed;
						
						//Następny krok
						iSimulationCase		:= 10;
						
					END_IF
				//Reset komendy ruchu osi X
				mcCartesianYMoveAbsolute.Execute		:= FALSE;
				
			END_IF
		END_IF	
				
		10:
			IF (CartesianZAxisRef.NcToPlc.ActPos > stParameters.lrTopZPosition - stParameters.lrBendingDistance) OR
				mcCartesianZMoveAbsolute.Done THEN
				//Jedź osią poziomą X na pozycję pick
				mcCartesianYMoveAbsolute.Execute		:= TRUE;
				mcCartesianYMoveAbsolute.Position		:= stParameters.lrPickYPosition;
				mcCartesianYMoveAbsolute.Acceleration	:= stParameters.lrPickerAcceleration;
				mcCartesianYMoveAbsolute.Deceleration	:= stParameters.lrPickerAcceleration;
				mcCartesianYMoveAbsolute.Velocity		:= stParameters.lrPickerSpeed;
				//Nakrętka pobrana z wózka nr.1
				bMover1InPickPos						:= SEL((stParameters.lrPickYPosition-GVL_Recipe.lrCapSorterPreScrewerPickXMover1PositionShow) <= 0.5, FALSE, TRUE);
				
				//Ustaw obracarkę w pozycji
				mcPreScrewerMoveRelative.Distance		:=  -1 * DINT_TO_LREAL((LREAL_TO_DINT(PreScrewerAxisRef.NcToPlc.SetPos)+diPreSCrewerHomePos) MOD 360);
				mcPreScrewerMoveRelative.Execute		:= mcPreScrewerMoveRelative.Distance<>0;
				mcPreScrewerMoveRelative.Acceleration	:= stParameters.lrScrewAcceleration;
				mcPreScrewerMoveRelative.Deceleration	:= stParameters.lrScrewAcceleration;
				mcPreScrewerMoveRelative.Velocity		:= stParameters.lrScrewSpeed;
			END_IF
			//Jak obie pozycje osiągnięte to wysuń chwytak słomek i następny krok
			IF mcCartesianYMoveAbsolute.Done AND mcCartesianZMoveAbsolute.Done AND mcCatcherMoveAbsolute.Done THEN
				IF mcPreScrewerMoveRelative.Done OR mcPreScrewerMoveRelative.Distance =0 THEN
					//Reset komendy ruchu osi
					mcCartesianYMoveAbsolute.Execute		:= FALSE;
					mcCartesianZMoveAbsolute.Execute		:= FALSE;
					mcPreScrewerMoveRelative.Execute		:= FALSE;
					mcCatcherMoveAbsolute.Execute			:= FALSE;
					//Wysuń chwytaki słomek jesli to potrzebuje recepta        
					bStrawCatcherActuatorIn					:= NOT stParameters.bStrawCatcherON;
					bStrawCatcherActuatorOut				:= stParameters.bStrawCatcherON;    
					//Następny krok
					iSimulationCase		:= 20;
				END_IF
			END_IF		
	
		20:
				mcCartesianZMoveAbsolute.Execute			:= TRUE;		
				mcCartesianZMoveAbsolute.Position			:= stParameters.lrPickZPosition;
				mcCartesianZMoveAbsolute.Acceleration		:= stParameters.lrPickerAcceleration;
				mcCartesianZMoveAbsolute.Deceleration		:= stParameters.lrPickerAcceleration;
				mcCartesianZMoveAbsolute.Velocity			:= stParameters.lrPickerSpeed;
					
			//Czekam na wykonanie ruchu
			IF mcCartesianZMoveAbsolute.Done THEN
				//Reset komendy ruchu osi
				mcCartesianZMoveAbsolute.Execute		:= FALSE;
				
				//Zeruje rejestry oraz załączanie ssawek
				 FOR i:=1 TO 4 DO
					 bCapSucker[i]						:= TRUE; 
					 aCapPresence[i] 					:= FALSE;					 
						IF stParameters.bPickerActiv[i] AND stParameters.bStrawCatcherON AND NOT stMoverStatus.stSlotStatus[i].bTubePresent THEN
							bReject								:= TRUE;
							bTubeReject							:= TRUE;
							lrAxisZ_RejectOffset				:= 0.0;
						END_IF
				 END_FOR
	    	
				//Następny krok
				iSimulationCase		:= 30;
			END_IF
	
		30:
			tonVacuumWatchdog.IN						:= TRUE;
		
			IF (tonSuckedOk[1].Q = stParameters.bPickerActiv[1] AND tonSuckedOk[2].Q = stParameters.bPickerActiv[2]
				AND tonSuckedOk[3].Q = stParameters.bPickerActiv[3] AND tonSuckedOk[4].Q = stParameters.bPickerActiv[4]) OR tonVacuumWatchdog.Q THEN
				tonVacuumWatchdog.IN					:= FALSE;
			
					FOR i:=1 TO 4 DO
						IF bMover1InPlacePos THEN
							diMover1VacuumRetry[i]		:= 0;
						ELSE
							diMover2VacuumRetry[i]		:= 0;
						END_IF	
					END_FOR 
					
				iSimulationCase		:= 40;
			END_IF	
			
		35:
			IF bReject THEN
				Reject();
				IF bRejectDone THEN				
					iSimulationCase					:= 0;	
				END_IF		
			ELSE
				iSimulationCase						:= 40;	
			END_IF	

		40:
			mcCartesianZMoveAbsolute.Execute		:= NOT stParameters.bVacuumDeactivate;		
			mcCartesianZMoveAbsolute.Position		:= stParameters.lrTopZPosition;
			mcCartesianZMoveAbsolute.Acceleration	:= SEL(GVL_Recipe.iCapSorterProductType = 0 ,stParameters.lrPickerAcceleration , 70.0);//stParameters.lrPickerAcceleration;
			mcCartesianZMoveAbsolute.Deceleration	:= stParameters.lrPickerAcceleration;
			mcCartesianZMoveAbsolute.Velocity		:= stParameters.lrPickerSpeed;
			tonCapCatcher.IN						:= FALSE;
			
				//przepisuje do rejestrów nakretki które kartezjan pobrał
			aCapPresence[1] := bCapSucker[1];
			aCapPresence[2] := bCapSucker[2];
			aCapPresence[3] := bCapSucker[3];
			aCapPresence[4] := bCapSucker[4];	
			
			IF mcCartesianZMoveAbsolute.Busy OR stParameters.bVacuumDeactivate THEN
				mcCartesianZMoveAbsolute.Execute		:= FALSE;
				iSimulationCase		:= 50;
			END_IF
		
		50:
				//Kleją się kulki 
			IF NOT stParameters.bVacuumDeactivate THEN					
				IF CartesianZAxisRef.NcToPlc.ActPos > stParameters.lrPickZPosition + 10.0 THEN
					mcCartesianZMoveAbsolute2.Execute		:= NOT stParameters.bVacuumDeactivate;		
					mcCartesianZMoveAbsolute2.Position		:= stParameters.lrTopZPosition;
					mcCartesianZMoveAbsolute2.Acceleration	:= stParameters.lrPickerAcceleration;
					mcCartesianZMoveAbsolute2.Deceleration	:= stParameters.lrPickerAcceleration;
					mcCartesianZMoveAbsolute2.Velocity		:= stParameters.lrPickerSpeed;
				END_IF
			END_IF

			IF CartesianZAxisRef.NcToPlc.ActPos > stParameters.lrCapCatcherZPosition OR (CartesianZAxisRef.NcToPlc.ActPos > stParameters.lrTopZPosition - 10) THEN
				bCapCatcher1							:= TRUE;
				bCapCatcher2							:= true;
				bCapCatcher3							:= true;
				bCapCatcher4							:= true;
				tonCapCatcher.IN						:= stParameters.bVacuumDeactivate;
			END_IF	
			
			mcCartesianZMoveAbsolute.Execute		:= tonCapCatcher.Q;	
			
			//Dodać sprawdzenie czy gotowy chwytak słomek !!!!!
			//Sprawdzenie pozycji osi pionowej Z i czy wysunięty siłownik chwytaka słomek
			IF ((CartesianZAxisRef.NcToPlc.ActPos > stParameters.lrTopZPosition - 10) OR
				mcCartesianZMoveAbsolute.Done) AND (tonStrawCatcherOut.Q OR NOT stParameters.bStrawCatcherON) THEN
				//Jedź osią poziomą X na pozycję pick
					mcCartesianZMoveAbsolute2.Execute		:= FALSE;
					bCapsBlowON								:= FALSE;
					iSimulationCase							:= 60;
					tonCapCatcher.IN						:= FALSE;
			END_IF
        	
		60:
			bCapCatcher1								:= TRUE;//bCapSucker1;
			bCapCatcher2								:= TRUE;//bCapSucker2;
			bCapCatcher3								:= TRUE;//bCapSucker3;
			bCapCatcher4								:= TRUE;//bCapSucker4;
	
			mcCartesianYMoveAbsolute.Position			:= 3.0;
			mcCartesianYMoveAbsolute.Acceleration		:= stParameters.lrPickerAcceleration;
			mcCartesianYMoveAbsolute.Deceleration		:= stParameters.lrPickerAcceleration;
			mcCartesianYMoveAbsolute.Velocity			:= stParameters.lrPickerSpeed;
			mcCartesianYMoveAbsolute.Execute			:= TRUE;
				
			IF CartesianYAxisRef.NcToPlc.ActPos < 40.0 THEN
				mcCartesianYMoveAbsolute.Execute		:= FALSE;
				iSimulationCase							:= 70;
			END_IF
			
			
			70:
				mcCartesianZMoveAbsolute.Execute			:= TRUE;		
				mcCartesianZMoveAbsolute.Position			:= 360;//stParameters.lrTopZPosition;
				mcCartesianZMoveAbsolute.Acceleration		:= stParameters.lrPickerAcceleration;
				mcCartesianZMoveAbsolute.Deceleration		:= stParameters.lrPickerAcceleration;
				mcCartesianZMoveAbsolute.Velocity			:= stParameters.lrPickerSpeed;
									
					IF mcCartesianZMoveAbsolute.Done THEN
						mcCartesianZMoveAbsolute.Execute	:= FALSE;	
							//Otwórz chwytaki
						bCapCatcher1						:= FALSE;
						bCapCatcher2						:= FALSE;
						bCapCatcher3						:= FALSE;
						bCapCatcher4						:= FALSE;
							//Wyłącz ssawki         		
						bCapSucker[1]						:= FALSE;
						bCapSucker[2]						:= FALSE;
						bCapSucker[3]						:= FALSE;
						bCapSucker[4]						:= FALSE;
						bCapsBlowON							:= TRUE;
						bCapBlow1 							:= TRUE;
						bCapBlow2 							:= TRUE;
						bCapBlow3 							:= TRUE;
						bCapBlow4 							:= TRUE;
						iSimulationCase						:= 80;
					END_IF
				
				80:
					mcCartesianZMoveAbsolute2.Execute		:= TRUE;		
					mcCartesianZMoveAbsolute2.Position		:= stParameters.lrTopZPosition;
					mcCartesianZMoveAbsolute2.Acceleration	:= stParameters.lrPickerAcceleration;
					mcCartesianZMoveAbsolute2.Deceleration	:= stParameters.lrPickerAcceleration;
					mcCartesianZMoveAbsolute2.Velocity		:= stParameters.lrPickerSpeed;
						
						IF 	mcCartesianZMoveAbsolute2.Done THEN
							mcCartesianZMoveAbsolute2.Execute	:= FALSE;
							iSimulationCase						:= 90;
						END_IF
			
				90:
					IF NOT bCapBlow1 AND NOT bCapBlow2 AND NOT bCapBlow3 AND NOT bCapBlow4 THEN
						mcCartesianYMoveAbsolute.Execute		:= TRUE;
						mcCartesianYMoveAbsolute.Position		:= stParameters.lrPickYPosition;
						mcCartesianYMoveAbsolute.Acceleration	:= stParameters.lrPickerAcceleration;
						mcCartesianYMoveAbsolute.Deceleration	:= stParameters.lrPickerAcceleration;
						mcCartesianYMoveAbsolute.Velocity		:= stParameters.lrPickerSpeed;
						iSimulationCase							:= 100;
					END_IF
			
				100:
					IF mcCartesianYMoveAbsolute.Done THEN
						mcCartesianYMoveAbsolute.Execute	:= FALSE;
						iSimulationCase						:= 0;
						bCycleDone							:= TRUE;
						eState								:= E_Station.eDone;
					END_IF

END_CASE
END_ACTION

END_FUNCTION_BLOCK

(* stored: Version 1.2.0.0, ProductVersion 3.1.4026.13, FileIdentifier 2fd00ac4ed79775e1e055d1ad5a79d17dfce516f, FileSignature 072e07333f89175ce09b147bb86dea810ff3829252c2360f384b109e59de71ed64d0cd9a639c074c09290934f8fecd30999f252f9145433e1091fdf7fc65c222fa408ed352e98a5f9f256760cde99c5ef5c3f7c77419d9110bc1cef0f0382971667baed0d4d23af6839833ef170fdd7d34443c933bf324390dede0939df8b209f23df8f297890e9e7e131d2547fa931c4f0ccec6a498cd4c9aefc7d8298e161d78fdf5bce67ae5eee6be1a4391d956fd3e650109b5bc552b1a80afe125fe6d54b3be73eef7fc7cac77533f307f034dd2ca07ee539e8621751f41fc21118a42b05c8c2c9539cf91c1787ba860acc809d8d45555c35432778a5171b8c1cd1b54df
   POU FB_CapPreScrewer: Id {8017741f-e68a-4a4b-856b-c4cf01a74f56}, SpecialFunc None
   Folder Running: Id {3dc13f7b-2ef8-4884-94d2-58057240c258}
   Action ACT_ErrorInit: Id {8ba1503a-97e6-4abe-8a1c-215cfe60f0b4}
   Action ACT_VirtualAxisControl: Id {5a0de19c-2e45-4d29-923f-b08186a2773c}
   Action ADS_Control: Id {7a872a3a-df41-43e9-b369-515f67b93f05}
   Action CamCalculation: Id {62126c6e-96c1-4c87-b94d-2c586899b486}
   Action CollisionAvoidance: Id {bcd2dc3e-bf23-4aad-b313-d3455f0f59cc}
   Action Control: Id {f3de3131-8318-40ed-89dc-8baf8da39b70}
   Action ErrorHandling: Id {874971a2-1f55-45d0-a322-9ff017616a3b}
   Action FBs: Id {5c006b73-ae1a-4890-8675-5320ba4c3b2e}
   Action Homing: Id {c4494d8c-b66c-4717-9939-5be64e011d7e}
   Action ManualMovements: Id {80bfc336-2e91-4102-930e-ae5e6c431cdd}
   Action PreparingToDisable: Id {9e509aa2-edad-4e76-acfc-006de33dcb11}
   Action Reject: Id {50e3cf8e-9904-431a-a0c5-d9e9045084aa}
   Action ResetCommands: Id {3945bcaa-decf-44a3-ab54-eb271aefcc05}
   Action Running: Id {7d334f5a-9797-4063-8f4d-7a8c0641b4b1}
   Action RunningCam: Id {6c98f202-d570-4f00-a619-dd30153f9542}
   Action RunningWithFlyingSaw: Id {82fe34a3-a77a-4611-94db-c4597230955b}
   Action Signals: Id {358b0970-a4f9-45ee-b951-6eab93c3d3ad}
   Action Simulation: Id {7fdb9db1-0fc8-4ed9-a791-b597c6693c3f} *)
